Universal Robots PolyScope program: interpreterModeSequential.urp

Program example1 (installation=default directory=/programs createdIn=5.10.0.1051222 lastSavedIn=5.10.0.1051222 robotSerialNumber=20175300007)
Robot Program (runOnlyOnce=true)
  Script: global exit_thread = False
  Script: interpreter_mode(clearOnEnd = False)
  Script: interpreter_mode()
